// Mitsubishi GX Works2 project: 0710-DA전압   PLC: Q02/Q02H

PROGRAM MAIN
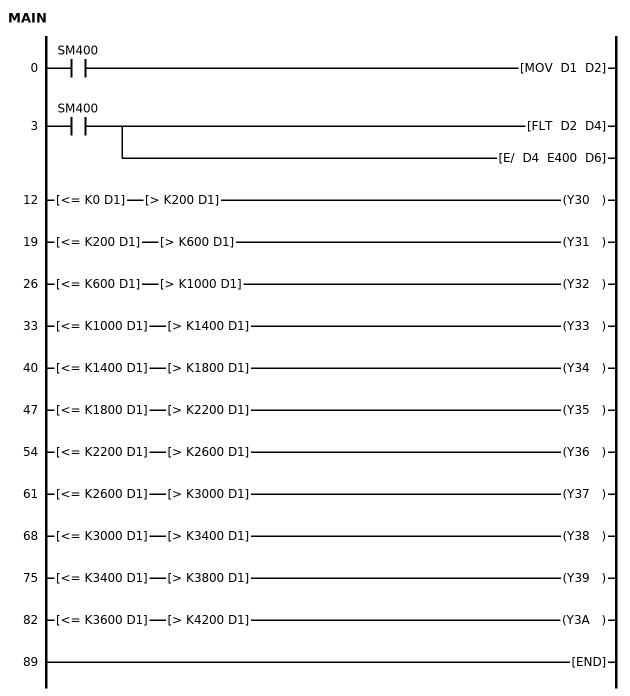
0     LD      SM400
      MOV     D1 D2
3     LD      SM400
      FLT     D2 D4
      E/      D4 E400 D6
12    LD<=    K0 D1
      AND>    K200 D1
      OUT     Y30
19    LD<=    K200 D1
      AND>    K600 D1
      OUT     Y31
26    LD<=    K600 D1
      AND>    K1000 D1
      OUT     Y32
33    LD<=    K1000 D1
      AND>    K1400 D1
      OUT     Y33
40    LD<=    K1400 D1
      AND>    K1800 D1
      OUT     Y34
47    LD<=    K1800 D1
      AND>    K2200 D1
      OUT     Y35
54    LD<=    K2200 D1
      AND>    K2600 D1
      OUT     Y36
61    LD<=    K2600 D1
      AND>    K3000 D1
      OUT     Y37
68    LD<=    K3000 D1
      AND>    K3400 D1
      OUT     Y38
75    LD<=    K3400 D1
      AND>    K3800 D1
      OUT     Y39
82    LD<=    K3600 D1
      AND>    K4200 D1
      OUT     Y3A
89    END
END_PROGRAM
